// TIA Portal V21 export
FUNCTION "BatchValves" : Void   // FC302, LAD
{ S7_Optimized_Access := 'TRUE' }
// stored: AutoNumber false, SetENOAutomatically false
BEGIN

REGION Network 1: ***************FILL WFI *****************
END_REGION

REGION Network 2: "BatchVessel".Cv02 ----- Wfi
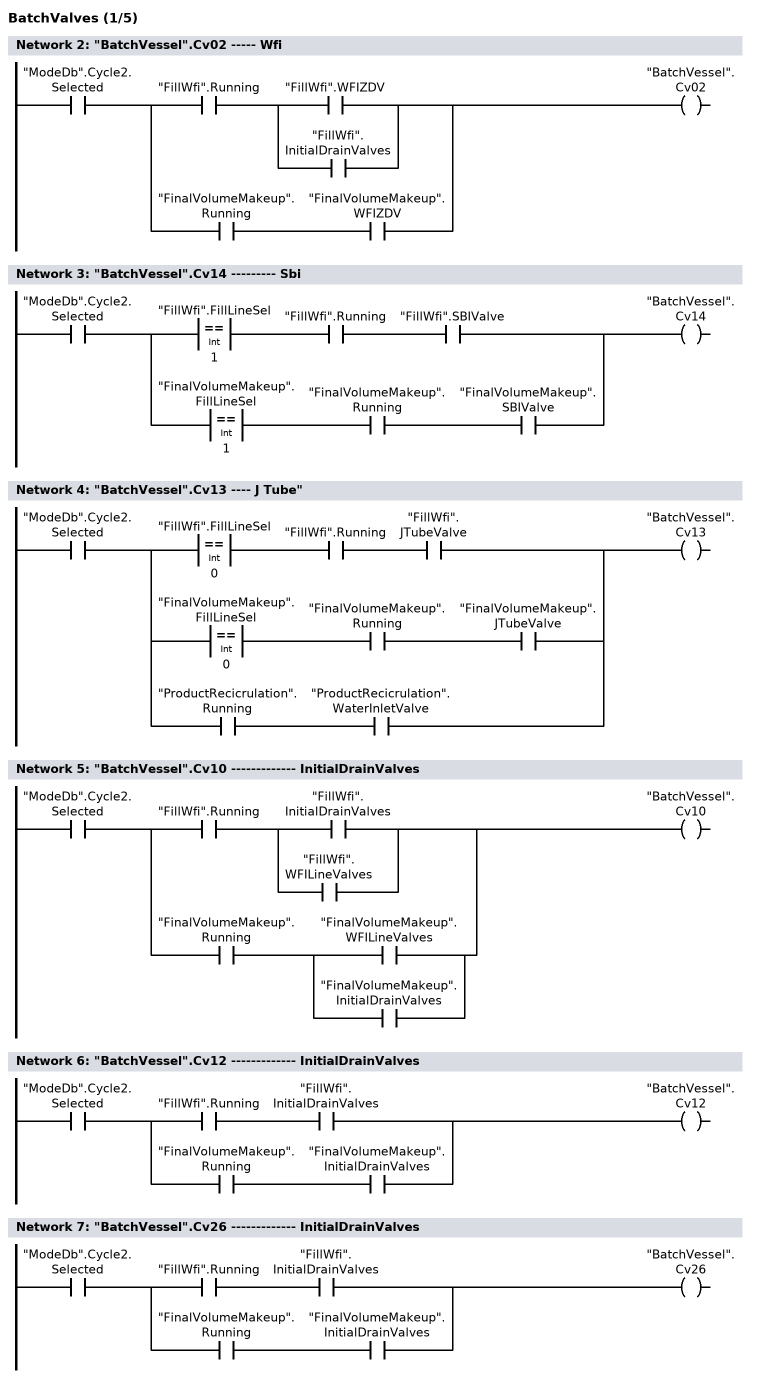
   RUNG wire#powerrail
      Contact( "ModeDb".Cycle2.Selected )
      wire#w1
      Contact( "FillWfi".Running )
      wire#w2
      Contact( "FillWfi".WFIZDV )
      wire#w3
      Coil( "BatchVessel".Cv02 )
   END_RUNG
   RUNG wire#w2
      Contact( "FillWfi".InitialDrainValves )
   END_RUNG wire#w3
   RUNG wire#w1
      Contact( "FinalVolumeMakeup".Running )
      Contact( "FinalVolumeMakeup".WFIZDV )
   END_RUNG wire#w3
   // the same network as SCL:
   "BatchVessel".Cv02 := "ModeDb".Cycle2.Selected AND (("FillWfi".Running AND ("FillWfi".WFIZDV OR "FillWfi".InitialDrainValves)) OR ("FinalVolumeMakeup".Running AND "FinalVolumeMakeup".WFIZDV));
END_REGION

REGION Network 3: "BatchVessel".Cv14 --------- Sbi
   RUNG wire#powerrail
      Contact( "ModeDb".Cycle2.Selected )
      wire#w1
      { S7_Templates := "SrcType := Int" } EQ_Contact(in1 := "FillWfi".FillLineSel, in2 := 1)
      Contact( "FillWfi".Running )
      Contact( "FillWfi".SBIValve )
      wire#w2
      Coil( "BatchVessel".Cv14 )
   END_RUNG
   RUNG wire#w1
      { S7_Templates := "SrcType := Int" } EQ_Contact(in1 := "FinalVolumeMakeup".FillLineSel, in2 := 1)
      Contact( "FinalVolumeMakeup".Running )
      Contact( "FinalVolumeMakeup".SBIValve )
   END_RUNG wire#w2
   // the same network as SCL:
   "BatchVessel".Cv14 := "ModeDb".Cycle2.Selected AND ((("FillWfi".FillLineSel = 1) AND "FillWfi".Running AND "FillWfi".SBIValve) OR (("FinalVolumeMakeup".FillLineSel = 1) AND "FinalVolumeMakeup".Running AND "FinalVolumeMakeup".SBIValve));
END_REGION

REGION Network 4: "BatchVessel".Cv13 ---- J Tube"
   RUNG wire#powerrail
      Contact( "ModeDb".Cycle2.Selected )
      wire#w1
      { S7_Templates := "SrcType := Int" } EQ_Contact(in1 := "FillWfi".FillLineSel, in2 := 0)
      Contact( "FillWfi".Running )
      Contact( "FillWfi".JTubeValve )
      wire#w2
      Coil( "BatchVessel".Cv13 )
   END_RUNG
   RUNG wire#w1
      { S7_Templates := "SrcType := Int" } EQ_Contact(in1 := "FinalVolumeMakeup".FillLineSel, in2 := 0)
      Contact( "FinalVolumeMakeup".Running )
      Contact( "FinalVolumeMakeup".JTubeValve )
   END_RUNG wire#w2
   RUNG wire#w1
      Contact( "ProductRecicrulation".Running )
      Contact( "ProductRecicrulation".WaterInletValve )
   END_RUNG wire#w2
   // the same network as SCL:
   "BatchVessel".Cv13 := "ModeDb".Cycle2.Selected AND ((("FillWfi".FillLineSel = 0) AND "FillWfi".Running AND "FillWfi".JTubeValve) OR (("FinalVolumeMakeup".FillLineSel = 0) AND "FinalVolumeMakeup".Running AND "FinalVolumeMakeup".JTubeValve) OR ("ProductRecicrulation".Running AND "ProductRecicrulation".WaterInletValve));
END_REGION

REGION Network 5: "BatchVessel".Cv10 ------------- InitialDrainValves
   RUNG wire#powerrail
      Contact( "ModeDb".Cycle2.Selected )
      wire#w1
      Contact( "FillWfi".Running )
      wire#w2
      Contact( "FillWfi".InitialDrainValves )
      wire#w3
      Coil( "BatchVessel".Cv10 )
   END_RUNG
   RUNG wire#w2
      Contact( "FillWfi".WFILineValves )
   END_RUNG wire#w3
   RUNG wire#w1
      Contact( "FinalVolumeMakeup".Running )
      wire#w4
      Contact( "FinalVolumeMakeup".WFILineValves )
   END_RUNG wire#w3
   RUNG wire#w4
      Contact( "FinalVolumeMakeup".InitialDrainValves )
   END_RUNG wire#w3
   // the same network as SCL:
   "BatchVessel".Cv10 := "ModeDb".Cycle2.Selected AND (("FillWfi".Running AND ("FillWfi".InitialDrainValves OR "FillWfi".WFILineValves)) OR ("FinalVolumeMakeup".Running AND ("FinalVolumeMakeup".WFILineValves OR "FinalVolumeMakeup".InitialDrainValves)));
END_REGION

REGION Network 6: "BatchVessel".Cv12 ------------- InitialDrainValves
   RUNG wire#powerrail
      Contact( "ModeDb".Cycle2.Selected )
      wire#w1
      Contact( "FillWfi".Running )
      Contact( "FillWfi".InitialDrainValves )
      wire#w2
      Coil( "BatchVessel".Cv12 )
   END_RUNG
   RUNG wire#w1
      Contact( "FinalVolumeMakeup".Running )
      Contact( "FinalVolumeMakeup".InitialDrainValves )
   END_RUNG wire#w2
   // the same network as SCL:
   "BatchVessel".Cv12 := "ModeDb".Cycle2.Selected AND (("FillWfi".Running AND "FillWfi".InitialDrainValves) OR ("FinalVolumeMakeup".Running AND "FinalVolumeMakeup".InitialDrainValves));
END_REGION

REGION Network 7: "BatchVessel".Cv26 ------------- InitialDrainValves
   RUNG wire#powerrail
      Contact( "ModeDb".Cycle2.Selected )
      wire#w1
      Contact( "FillWfi".Running )
      Contact( "FillWfi".InitialDrainValves )
      wire#w2
      Coil( "BatchVessel".Cv26 )
   END_RUNG
   RUNG wire#w1
      Contact( "FinalVolumeMakeup".Running )
      Contact( "FinalVolumeMakeup".InitialDrainValves )
   END_RUNG wire#w2
   // the same network as SCL:
   "BatchVessel".Cv26 := "ModeDb".Cycle2.Selected AND (("FillWfi".Running AND "FillWfi".InitialDrainValves) OR ("FinalVolumeMakeup".Running AND "FinalVolumeMakeup".InitialDrainValves));
END_REGION

REGION Network 8: "BatchVessel".Fbov01 ------------- InitialDrainValves
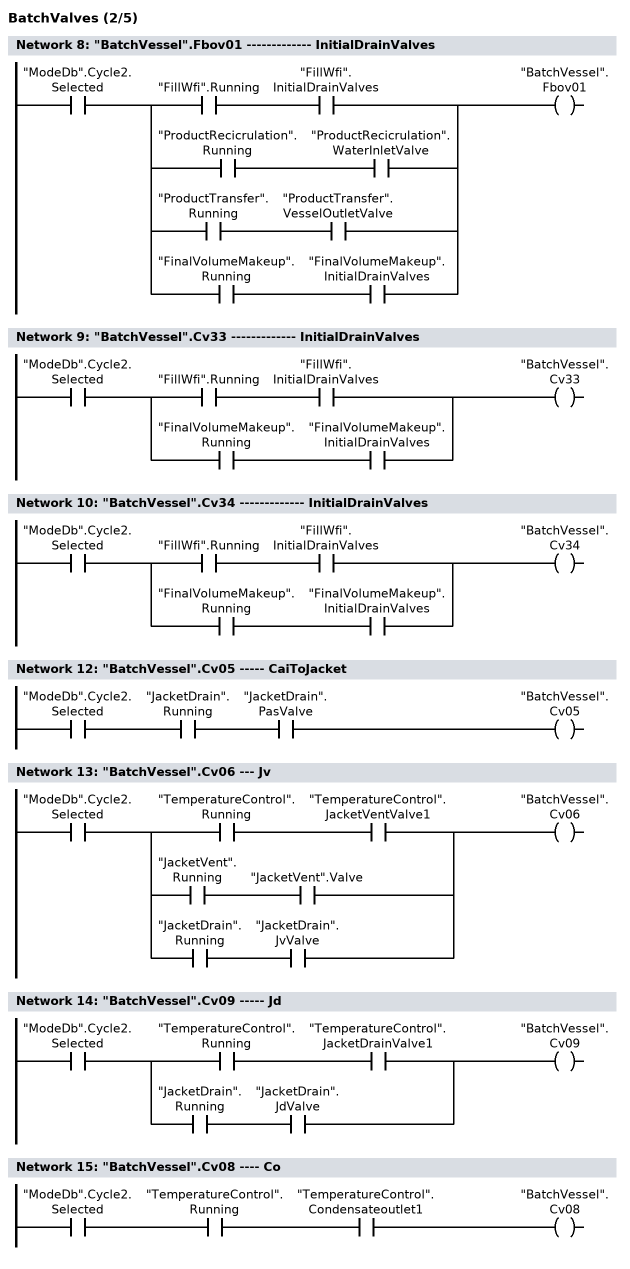
   RUNG wire#powerrail
      Contact( "ModeDb".Cycle2.Selected )
      wire#w1
      Contact( "FillWfi".Running )
      Contact( "FillWfi".InitialDrainValves )
      wire#w2
      Coil( "BatchVessel".Fbov01 )
   END_RUNG
   RUNG wire#w1
      Contact( "ProductRecicrulation".Running )
      Contact( "ProductRecicrulation".WaterInletValve )
   END_RUNG wire#w2
   RUNG wire#w1
      Contact( "ProductTransfer".Running )
      Contact( "ProductTransfer".VesselOutletValve )
   END_RUNG wire#w2
   RUNG wire#w1
      Contact( "FinalVolumeMakeup".Running )
      Contact( "FinalVolumeMakeup".InitialDrainValves )
   END_RUNG wire#w2
   // the same network as SCL:
   "BatchVessel".Fbov01 := "ModeDb".Cycle2.Selected AND (("FillWfi".Running AND "FillWfi".InitialDrainValves) OR ("ProductRecicrulation".Running AND "ProductRecicrulation".WaterInletValve) OR ("ProductTransfer".Running AND "ProductTransfer".VesselOutletValve) OR ("FinalVolumeMakeup".Running AND "FinalVolumeMakeup".InitialDrainValves));
END_REGION

REGION Network 9: "BatchVessel".Cv33 ------------- InitialDrainValves
   RUNG wire#powerrail
      Contact( "ModeDb".Cycle2.Selected )
      wire#w1
      Contact( "FillWfi".Running )
      Contact( "FillWfi".InitialDrainValves )
      wire#w2
      Coil( "BatchVessel".Cv33 )
   END_RUNG
   RUNG wire#w1
      Contact( "FinalVolumeMakeup".Running )
      Contact( "FinalVolumeMakeup".InitialDrainValves )
   END_RUNG wire#w2
   // the same network as SCL:
   "BatchVessel".Cv33 := "ModeDb".Cycle2.Selected AND (("FillWfi".Running AND "FillWfi".InitialDrainValves) OR ("FinalVolumeMakeup".Running AND "FinalVolumeMakeup".InitialDrainValves));
END_REGION

REGION Network 10: "BatchVessel".Cv34 ------------- InitialDrainValves
   RUNG wire#powerrail
      Contact( "ModeDb".Cycle2.Selected )
      wire#w1
      Contact( "FillWfi".Running )
      Contact( "FillWfi".InitialDrainValves )
      wire#w2
      Coil( "BatchVessel".Cv34 )
   END_RUNG
   RUNG wire#w1
      Contact( "FinalVolumeMakeup".Running )
      Contact( "FinalVolumeMakeup".InitialDrainValves )
   END_RUNG wire#w2
   // the same network as SCL:
   "BatchVessel".Cv34 := "ModeDb".Cycle2.Selected AND (("FillWfi".Running AND "FillWfi".InitialDrainValves) OR ("FinalVolumeMakeup".Running AND "FinalVolumeMakeup".InitialDrainValves));
END_REGION

REGION Network 11: ***************TEMPERATURE CONTROL *****************
END_REGION

REGION Network 12: "BatchVessel".Cv05 ----- CaiToJacket
   RUNG wire#powerrail
      Contact( "ModeDb".Cycle2.Selected )
      Contact( "JacketDrain".Running )
      Contact( "JacketDrain".PasValve )
      Coil( "BatchVessel".Cv05 )
   END_RUNG
   // the same network as SCL:
   "BatchVessel".Cv05 := "ModeDb".Cycle2.Selected AND "JacketDrain".Running AND "JacketDrain".PasValve;
END_REGION

REGION Network 13: "BatchVessel".Cv06 --- Jv
   RUNG wire#powerrail
      Contact( "ModeDb".Cycle2.Selected )
      wire#w1
      Contact( "TemperatureControl".Running )
      Contact( "TemperatureControl".JacketVentValve1 )
      wire#w2
      Coil( "BatchVessel".Cv06 )
   END_RUNG
   RUNG wire#w1
      Contact( "JacketVent".Running )
      Contact( "JacketVent".Valve )
   END_RUNG wire#w2
   RUNG wire#w1
      Contact( "JacketDrain".Running )
      Contact( "JacketDrain".JvValve )
   END_RUNG wire#w2
   // the same network as SCL:
   "BatchVessel".Cv06 := "ModeDb".Cycle2.Selected AND (("TemperatureControl".Running AND "TemperatureControl".JacketVentValve1) OR ("JacketVent".Running AND "JacketVent".Valve) OR ("JacketDrain".Running AND "JacketDrain".JvValve));
END_REGION

REGION Network 14: "BatchVessel".Cv09 ----- Jd
   RUNG wire#powerrail
      Contact( "ModeDb".Cycle2.Selected )
      wire#w1
      Contact( "TemperatureControl".Running )
      Contact( "TemperatureControl".JacketDrainValve1 )
      wire#w2
      Coil( "BatchVessel".Cv09 )
   END_RUNG
   RUNG wire#w1
      Contact( "JacketDrain".Running )
      Contact( "JacketDrain".JdValve )
   END_RUNG wire#w2
   // the same network as SCL:
   "BatchVessel".Cv09 := "ModeDb".Cycle2.Selected AND (("TemperatureControl".Running AND "TemperatureControl".JacketDrainValve1) OR ("JacketDrain".Running AND "JacketDrain".JdValve));
END_REGION

REGION Network 15: "BatchVessel".Cv08 ---- Co
   RUNG wire#powerrail
      Contact( "ModeDb".Cycle2.Selected )
      Contact( "TemperatureControl".Running )
      Contact( "TemperatureControl".Condensateoutlet1 )
      Coil( "BatchVessel".Cv08 )
   END_RUNG
   // the same network as SCL:
   "BatchVessel".Cv08 := "ModeDb".Cycle2.Selected AND "TemperatureControl".Running AND "TemperatureControl".Condensateoutlet1;
END_REGION

REGION Network 16: "BatchVessel".Cv04 ---- Psi
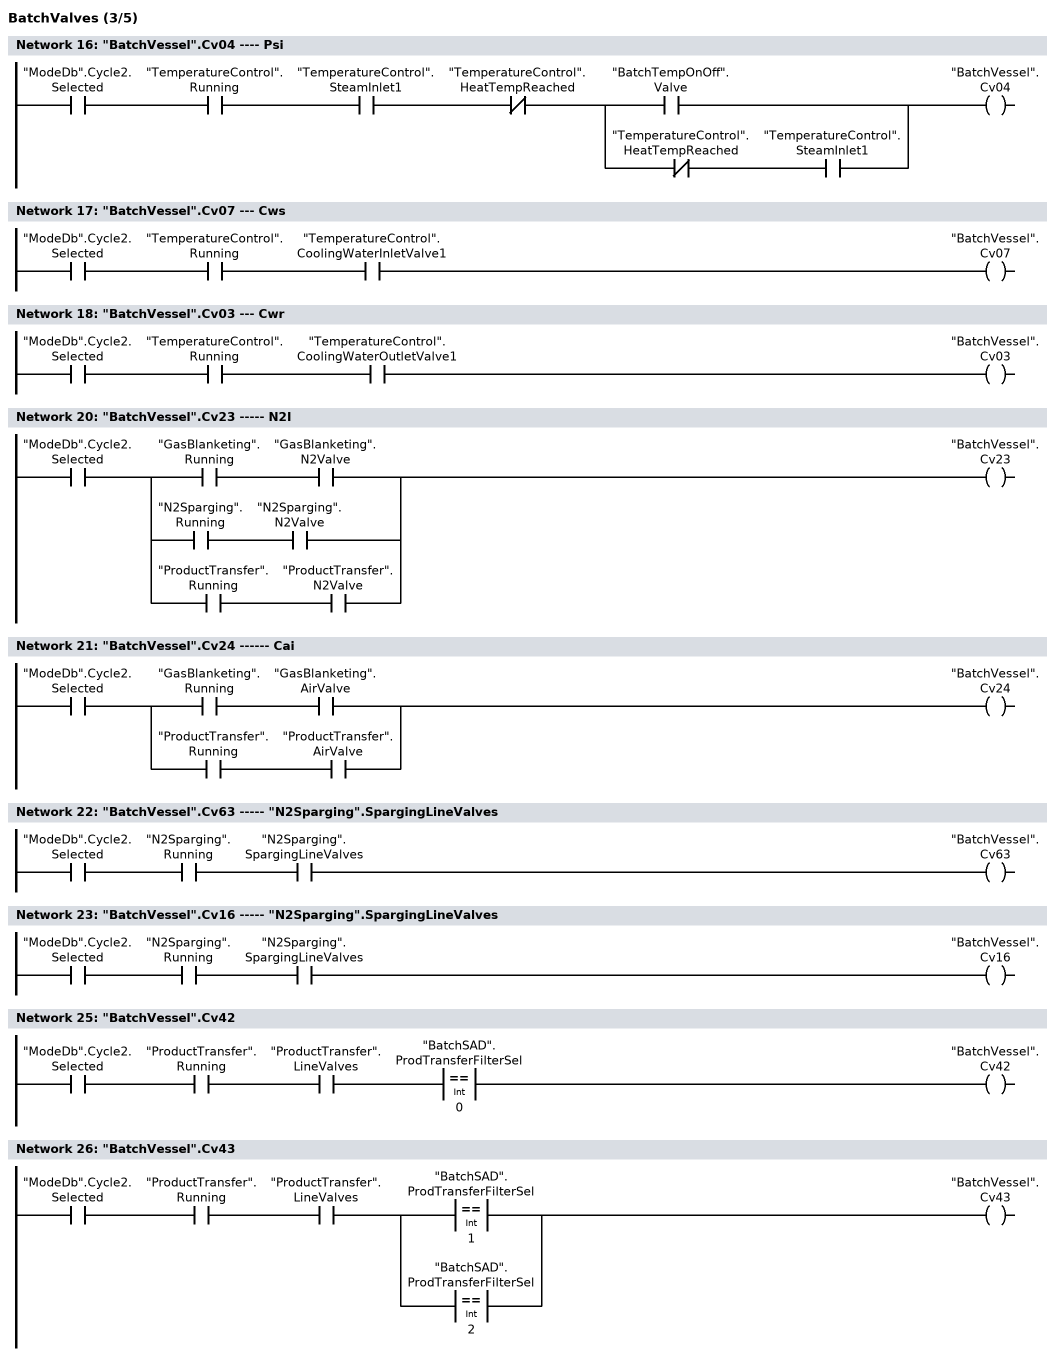
   RUNG wire#powerrail
      Contact( "ModeDb".Cycle2.Selected )
      Contact( "TemperatureControl".Running )
      Contact( "TemperatureControl".SteamInlet1 )
      I_Contact( "TemperatureControl".HeatTempReached )
      wire#w1
      Contact( "BatchTempOnOff".Valve )
      wire#w2
      Coil( "BatchVessel".Cv04 )
   END_RUNG
   RUNG wire#w1
      I_Contact( "TemperatureControl".HeatTempReached )
      Contact( "TemperatureControl".SteamInlet1 )
   END_RUNG wire#w2
   // the same network as SCL:
   "BatchVessel".Cv04 := "ModeDb".Cycle2.Selected AND "TemperatureControl".Running AND "TemperatureControl".SteamInlet1 AND NOT "TemperatureControl".HeatTempReached AND ("BatchTempOnOff".Valve OR (NOT "TemperatureControl".HeatTempReached AND "TemperatureControl".SteamInlet1));
END_REGION

REGION Network 17: "BatchVessel".Cv07 --- Cws
   RUNG wire#powerrail
      Contact( "ModeDb".Cycle2.Selected )
      Contact( "TemperatureControl".Running )
      Contact( "TemperatureControl".CoolingWaterInletValve1 )
      Coil( "BatchVessel".Cv07 )
   END_RUNG
   // the same network as SCL:
   "BatchVessel".Cv07 := "ModeDb".Cycle2.Selected AND "TemperatureControl".Running AND "TemperatureControl".CoolingWaterInletValve1;
END_REGION

REGION Network 18: "BatchVessel".Cv03 --- Cwr
   RUNG wire#powerrail
      Contact( "ModeDb".Cycle2.Selected )
      Contact( "TemperatureControl".Running )
      Contact( "TemperatureControl".CoolingWaterOutletValve1 )
      Coil( "BatchVessel".Cv03 )
   END_RUNG
   // the same network as SCL:
   "BatchVessel".Cv03 := "ModeDb".Cycle2.Selected AND "TemperatureControl".Running AND "TemperatureControl".CoolingWaterOutletValve1;
END_REGION

REGION Network 19: ***************GAS BLANKETING********N2 SPARGING*********
END_REGION

REGION Network 20: "BatchVessel".Cv23 ----- N2I
   RUNG wire#powerrail
      Contact( "ModeDb".Cycle2.Selected )
      wire#w1
      Contact( "GasBlanketing".Running )
      Contact( "GasBlanketing".N2Valve )
      wire#w2
      Coil( "BatchVessel".Cv23 )
   END_RUNG
   RUNG wire#w1
      Contact( "N2Sparging".Running )
      Contact( "N2Sparging".N2Valve )
   END_RUNG wire#w2
   RUNG wire#w1
      Contact( "ProductTransfer".Running )
      Contact( "ProductTransfer".N2Valve )
   END_RUNG wire#w2
   // the same network as SCL:
   "BatchVessel".Cv23 := "ModeDb".Cycle2.Selected AND (("GasBlanketing".Running AND "GasBlanketing".N2Valve) OR ("N2Sparging".Running AND "N2Sparging".N2Valve) OR ("ProductTransfer".Running AND "ProductTransfer".N2Valve));
END_REGION

REGION Network 21: "BatchVessel".Cv24 ------ Cai
   RUNG wire#powerrail
      Contact( "ModeDb".Cycle2.Selected )
      wire#w1
      Contact( "GasBlanketing".Running )
      Contact( "GasBlanketing".AirValve )
      wire#w2
      Coil( "BatchVessel".Cv24 )
   END_RUNG
   RUNG wire#w1
      Contact( "ProductTransfer".Running )
      Contact( "ProductTransfer".AirValve )
   END_RUNG wire#w2
   // the same network as SCL:
   "BatchVessel".Cv24 := "ModeDb".Cycle2.Selected AND (("GasBlanketing".Running AND "GasBlanketing".AirValve) OR ("ProductTransfer".Running AND "ProductTransfer".AirValve));
END_REGION

REGION Network 22: "BatchVessel".Cv63 ----- "N2Sparging".SpargingLineValves
   RUNG wire#powerrail
      Contact( "ModeDb".Cycle2.Selected )
      Contact( "N2Sparging".Running )
      Contact( "N2Sparging".SpargingLineValves )
      Coil( "BatchVessel".Cv63 )
   END_RUNG
   // the same network as SCL:
   "BatchVessel".Cv63 := "ModeDb".Cycle2.Selected AND "N2Sparging".Running AND "N2Sparging".SpargingLineValves;
END_REGION

REGION Network 23: "BatchVessel".Cv16 ----- "N2Sparging".SpargingLineValves
   RUNG wire#powerrail
      Contact( "ModeDb".Cycle2.Selected )
      Contact( "N2Sparging".Running )
      Contact( "N2Sparging".SpargingLineValves )
      Coil( "BatchVessel".Cv16 )
   END_RUNG
   // the same network as SCL:
   "BatchVessel".Cv16 := "ModeDb".Cycle2.Selected AND "N2Sparging".Running AND "N2Sparging".SpargingLineValves;
END_REGION

REGION Network 24: ***************PRODUCT TRANSFER*****************
END_REGION

REGION Network 25: "BatchVessel".Cv42
   RUNG wire#powerrail
      Contact( "ModeDb".Cycle2.Selected )
      Contact( "ProductTransfer".Running )
      Contact( "ProductTransfer".LineValves )
      { S7_Templates := "SrcType := Int" } EQ_Contact(in1 := "BatchSAD".ProdTransferFilterSel, in2 := 0)
      Coil( "BatchVessel".Cv42 )
   END_RUNG
   // the same network as SCL:
   "BatchVessel".Cv42 := "ModeDb".Cycle2.Selected AND "ProductTransfer".Running AND "ProductTransfer".LineValves AND ("BatchSAD".ProdTransferFilterSel = 0);
END_REGION

REGION Network 26: "BatchVessel".Cv43
   RUNG wire#powerrail
      Contact( "ModeDb".Cycle2.Selected )
      Contact( "ProductTransfer".Running )
      Contact( "ProductTransfer".LineValves )
      wire#w1
      { S7_Templates := "SrcType := Int" } EQ_Contact(in1 := "BatchSAD".ProdTransferFilterSel, in2 := 1)
      wire#w2
      Coil( "BatchVessel".Cv43 )
   END_RUNG
   RUNG wire#w1
      { S7_Templates := "SrcType := Int" } EQ_Contact(in1 := "BatchSAD".ProdTransferFilterSel, in2 := 2)
   END_RUNG wire#w2
   // the same network as SCL:
   "BatchVessel".Cv43 := "ModeDb".Cycle2.Selected AND "ProductTransfer".Running AND "ProductTransfer".LineValves AND (("BatchSAD".ProdTransferFilterSel = 1) OR ("BatchSAD".ProdTransferFilterSel = 2));
END_REGION

REGION Network 27: "BatchVessel".Cv48
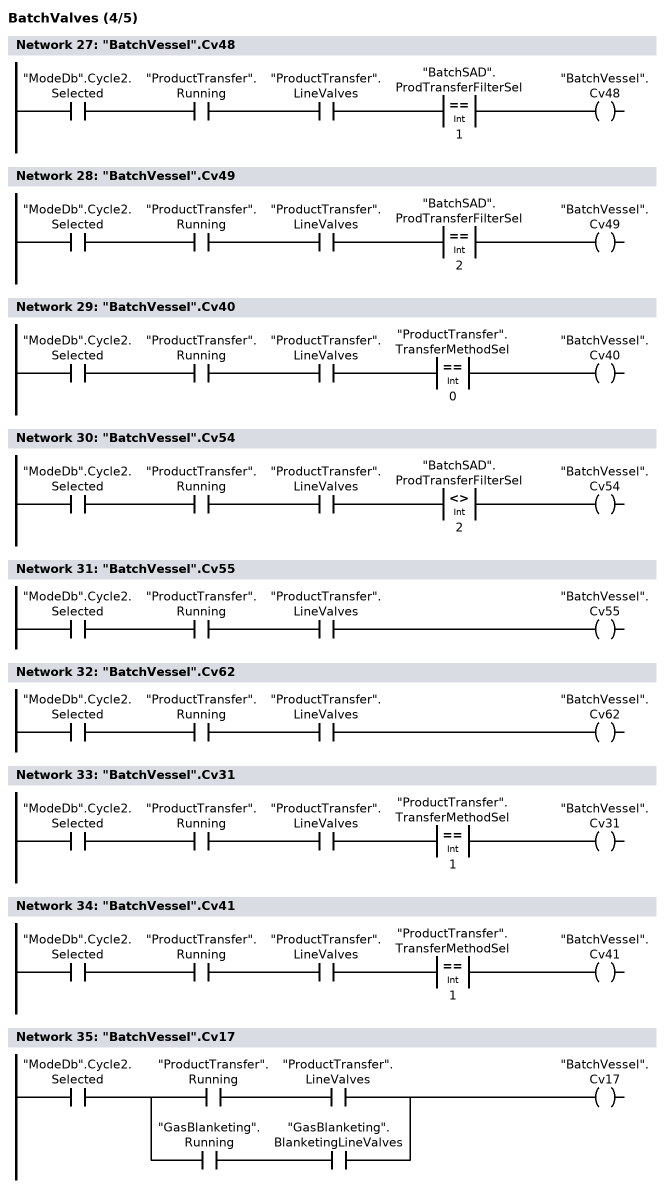
   RUNG wire#powerrail
      Contact( "ModeDb".Cycle2.Selected )
      Contact( "ProductTransfer".Running )
      Contact( "ProductTransfer".LineValves )
      { S7_Templates := "SrcType := Int" } EQ_Contact(in1 := "BatchSAD".ProdTransferFilterSel, in2 := 1)
      Coil( "BatchVessel".Cv48 )
   END_RUNG
   // the same network as SCL:
   "BatchVessel".Cv48 := "ModeDb".Cycle2.Selected AND "ProductTransfer".Running AND "ProductTransfer".LineValves AND ("BatchSAD".ProdTransferFilterSel = 1);
END_REGION

REGION Network 28: "BatchVessel".Cv49
   RUNG wire#powerrail
      Contact( "ModeDb".Cycle2.Selected )
      Contact( "ProductTransfer".Running )
      Contact( "ProductTransfer".LineValves )
      { S7_Templates := "SrcType := Int" } EQ_Contact(in1 := "BatchSAD".ProdTransferFilterSel, in2 := 2)
      Coil( "BatchVessel".Cv49 )
   END_RUNG
   // the same network as SCL:
   "BatchVessel".Cv49 := "ModeDb".Cycle2.Selected AND "ProductTransfer".Running AND "ProductTransfer".LineValves AND ("BatchSAD".ProdTransferFilterSel = 2);
END_REGION

REGION Network 29: "BatchVessel".Cv40
   RUNG wire#powerrail
      Contact( "ModeDb".Cycle2.Selected )
      Contact( "ProductTransfer".Running )
      Contact( "ProductTransfer".LineValves )
      { S7_Templates := "SrcType := Int" } EQ_Contact(in1 := "ProductTransfer".TransferMethodSel, in2 := 0)
      Coil( "BatchVessel".Cv40 )
   END_RUNG
   // the same network as SCL:
   "BatchVessel".Cv40 := "ModeDb".Cycle2.Selected AND "ProductTransfer".Running AND "ProductTransfer".LineValves AND ("ProductTransfer".TransferMethodSel = 0);
END_REGION

REGION Network 30: "BatchVessel".Cv54
   RUNG wire#powerrail
      Contact( "ModeDb".Cycle2.Selected )
      Contact( "ProductTransfer".Running )
      Contact( "ProductTransfer".LineValves )
      { S7_Templates := "SrcType := Int" } NE_Contact(in1 := "BatchSAD".ProdTransferFilterSel, in2 := 2)
      Coil( "BatchVessel".Cv54 )
   END_RUNG
   // the same network as SCL:
   "BatchVessel".Cv54 := "ModeDb".Cycle2.Selected AND "ProductTransfer".Running AND "ProductTransfer".LineValves AND ("BatchSAD".ProdTransferFilterSel <> 2);
END_REGION

REGION Network 31: "BatchVessel".Cv55
   RUNG wire#powerrail
      Contact( "ModeDb".Cycle2.Selected )
      Contact( "ProductTransfer".Running )
      Contact( "ProductTransfer".LineValves )
      Coil( "BatchVessel".Cv55 )
   END_RUNG
   // the same network as SCL:
   "BatchVessel".Cv55 := "ModeDb".Cycle2.Selected AND "ProductTransfer".Running AND "ProductTransfer".LineValves;
END_REGION

REGION Network 32: "BatchVessel".Cv62
   RUNG wire#powerrail
      Contact( "ModeDb".Cycle2.Selected )
      Contact( "ProductTransfer".Running )
      Contact( "ProductTransfer".LineValves )
      Coil( "BatchVessel".Cv62 )
   END_RUNG
   // the same network as SCL:
   "BatchVessel".Cv62 := "ModeDb".Cycle2.Selected AND "ProductTransfer".Running AND "ProductTransfer".LineValves;
END_REGION

REGION Network 33: "BatchVessel".Cv31
   RUNG wire#powerrail
      Contact( "ModeDb".Cycle2.Selected )
      Contact( "ProductTransfer".Running )
      Contact( "ProductTransfer".LineValves )
      { S7_Templates := "SrcType := Int" } EQ_Contact(in1 := "ProductTransfer".TransferMethodSel, in2 := 1)
      Coil( "BatchVessel".Cv31 )
   END_RUNG
   // the same network as SCL:
   "BatchVessel".Cv31 := "ModeDb".Cycle2.Selected AND "ProductTransfer".Running AND "ProductTransfer".LineValves AND ("ProductTransfer".TransferMethodSel = 1);
END_REGION

REGION Network 34: "BatchVessel".Cv41
   RUNG wire#powerrail
      Contact( "ModeDb".Cycle2.Selected )
      Contact( "ProductTransfer".Running )
      Contact( "ProductTransfer".LineValves )
      { S7_Templates := "SrcType := Int" } EQ_Contact(in1 := "ProductTransfer".TransferMethodSel, in2 := 1)
      Coil( "BatchVessel".Cv41 )
   END_RUNG
   // the same network as SCL:
   "BatchVessel".Cv41 := "ModeDb".Cycle2.Selected AND "ProductTransfer".Running AND "ProductTransfer".LineValves AND ("ProductTransfer".TransferMethodSel = 1);
END_REGION

REGION Network 35: "BatchVessel".Cv17
   RUNG wire#powerrail
      Contact( "ModeDb".Cycle2.Selected )
      wire#w1
      Contact( "ProductTransfer".Running )
      Contact( "ProductTransfer".LineValves )
      wire#w2
      Coil( "BatchVessel".Cv17 )
   END_RUNG
   RUNG wire#w1
      Contact( "GasBlanketing".Running )
      Contact( "GasBlanketing".BlanketingLineValves )
   END_RUNG wire#w2
   // the same network as SCL:
   "BatchVessel".Cv17 := "ModeDb".Cycle2.Selected AND (("ProductTransfer".Running AND "ProductTransfer".LineValves) OR ("GasBlanketing".Running AND "GasBlanketing".BlanketingLineValves));
END_REGION

REGION Network 36: ***************RM ADDITION*****************
END_REGION

REGION Network 37: "BatchVessel".Cv21 ---- Vent
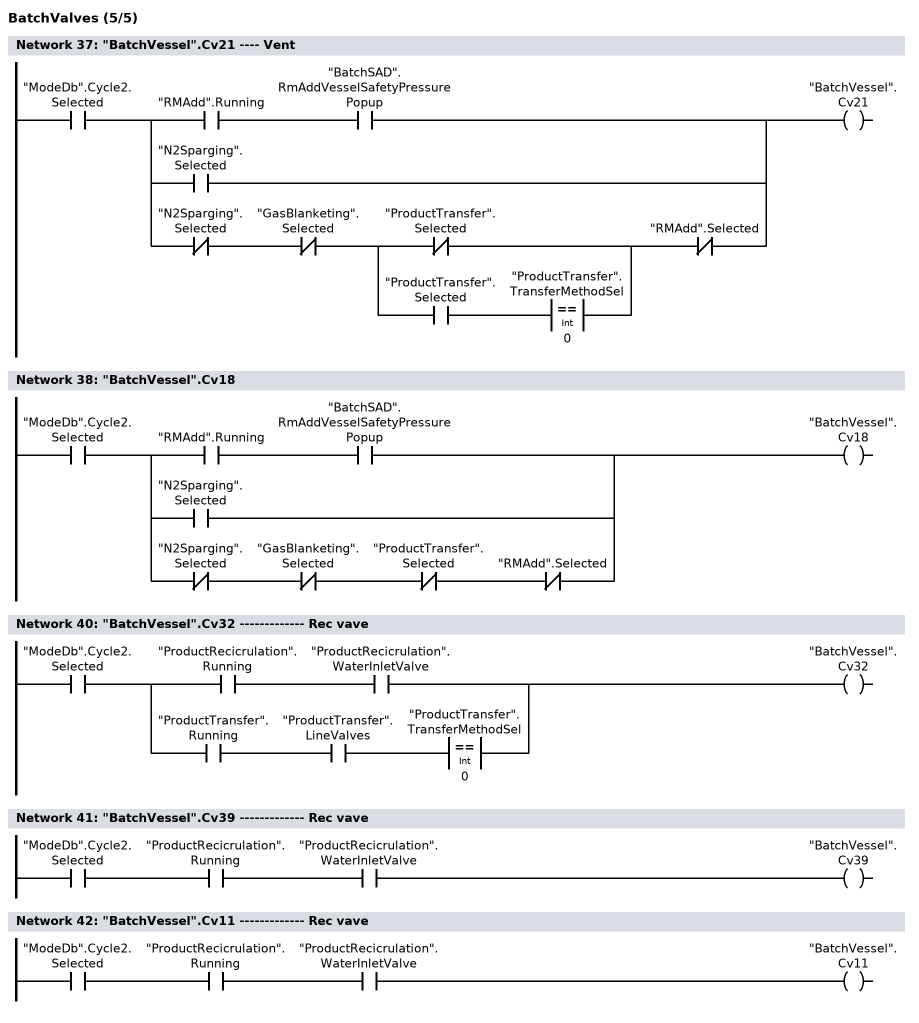
   RUNG wire#powerrail
      Contact( "ModeDb".Cycle2.Selected )
      wire#w1
      Contact( "RMAdd".Running )
      Contact( "BatchSAD".RmAddVesselSafetyPressurePopup )
      wire#w2
      Coil( "BatchVessel".Cv21 )
   END_RUNG
   RUNG wire#w1
      Contact( "N2Sparging".Selected )
   END_RUNG wire#w2
   RUNG wire#w1
      I_Contact( "N2Sparging".Selected )
      I_Contact( "GasBlanketing".Selected )
      wire#w3
      I_Contact( "ProductTransfer".Selected )
      wire#w4
      I_Contact( "RMAdd".Selected )
   END_RUNG wire#w2
   RUNG wire#w3
      Contact( "ProductTransfer".Selected )
      { S7_Templates := "SrcType := Int" } EQ_Contact(in1 := "ProductTransfer".TransferMethodSel, in2 := 0)
   END_RUNG wire#w4
   // the same network as SCL:
   "BatchVessel".Cv21 := "ModeDb".Cycle2.Selected AND (("RMAdd".Running AND "BatchSAD".RmAddVesselSafetyPressurePopup) OR "N2Sparging".Selected OR (NOT "N2Sparging".Selected AND NOT "GasBlanketing".Selected AND (NOT "ProductTransfer".Selected OR ("ProductTransfer".Selected AND ("ProductTransfer".TransferMethodSel = 0))) AND NOT "RMAdd".Selected));
END_REGION

REGION Network 38: "BatchVessel".Cv18
   RUNG wire#powerrail
      Contact( "ModeDb".Cycle2.Selected )
      wire#w1
      Contact( "RMAdd".Running )
      Contact( "BatchSAD".RmAddVesselSafetyPressurePopup )
      wire#w2
      Coil( "BatchVessel".Cv18 )
   END_RUNG
   RUNG wire#w1
      Contact( "N2Sparging".Selected )
   END_RUNG wire#w2
   RUNG wire#w1
      I_Contact( "N2Sparging".Selected )
      I_Contact( "GasBlanketing".Selected )
      I_Contact( "ProductTransfer".Selected )
      I_Contact( "RMAdd".Selected )
   END_RUNG wire#w2
   // the same network as SCL:
   "BatchVessel".Cv18 := "ModeDb".Cycle2.Selected AND (("RMAdd".Running AND "BatchSAD".RmAddVesselSafetyPressurePopup) OR "N2Sparging".Selected OR (NOT "N2Sparging".Selected AND NOT "GasBlanketing".Selected AND NOT "ProductTransfer".Selected AND NOT "RMAdd".Selected));
END_REGION

REGION Network 39: *************** PRODUCT RECIRCULATION *****************
END_REGION

REGION Network 40: "BatchVessel".Cv32 ------------- Rec vave
   RUNG wire#powerrail
      Contact( "ModeDb".Cycle2.Selected )
      wire#w1
      Contact( "ProductRecicrulation".Running )
      Contact( "ProductRecicrulation".WaterInletValve )
      wire#w2
      Coil( "BatchVessel".Cv32 )
   END_RUNG
   RUNG wire#w1
      Contact( "ProductTransfer".Running )
      Contact( "ProductTransfer".LineValves )
      { S7_Templates := "SrcType := Int" } EQ_Contact(in1 := "ProductTransfer".TransferMethodSel, in2 := 0)
   END_RUNG wire#w2
   // the same network as SCL:
   "BatchVessel".Cv32 := "ModeDb".Cycle2.Selected AND (("ProductRecicrulation".Running AND "ProductRecicrulation".WaterInletValve) OR ("ProductTransfer".Running AND "ProductTransfer".LineValves AND ("ProductTransfer".TransferMethodSel = 0)));
END_REGION

REGION Network 41: "BatchVessel".Cv39 ------------- Rec vave
   RUNG wire#powerrail
      Contact( "ModeDb".Cycle2.Selected )
      Contact( "ProductRecicrulation".Running )
      Contact( "ProductRecicrulation".WaterInletValve )
      Coil( "BatchVessel".Cv39 )
   END_RUNG
   // the same network as SCL:
   "BatchVessel".Cv39 := "ModeDb".Cycle2.Selected AND "ProductRecicrulation".Running AND "ProductRecicrulation".WaterInletValve;
END_REGION

REGION Network 42: "BatchVessel".Cv11 ------------- Rec vave
   RUNG wire#powerrail
      Contact( "ModeDb".Cycle2.Selected )
      Contact( "ProductRecicrulation".Running )
      Contact( "ProductRecicrulation".WaterInletValve )
      Coil( "BatchVessel".Cv11 )
   END_RUNG
   // the same network as SCL:
   "BatchVessel".Cv11 := "ModeDb".Cycle2.Selected AND "ProductRecicrulation".Running AND "ProductRecicrulation".WaterInletValve;
END_REGION
END_FUNCTION
